# EPICS substitutions: apps/jscalerApp/Db/jscalers_TDCFTOF5_TRIG.substitutions
file "db/jscaler_channel.db" {
pattern { CrNo,CrName,Sl,Ch,Det,Sys,Element,CScode,Thresh,Mode,Counts }
{ "05","TDCFTOF5","20","15","TRIG","DISC","SEC5_F00","5125","15","271","15" }
}
